TYPE ST_PIZZA :
STRUCT
	bExist : BOOL;
	dtTimeEnteredOven : DT;
	dtTimeExitedOven : DT;
	tTimeInOven : TIME;
	eType : E_PIZZA_TYPES;	// 0 - cheese, 1 - pepperoni, 2 - olives
END_STRUCT
END_TYPE

(* stored: Version 1.1.0.1, ProductVersion 3.1.4024.12
   DUT ST_PIZZA: Id {11b30019-a794-47eb-bc0a-2a4866c7c186} *)
